PROGRAM PRG_SFLX_NoValidationCamera
VAR
	rtrigValidCameraTrigger				: F_TRIG;
	bSideFlexValidCameraTrigger			: BOOL;

	rsSideFlexTwoOutersInAggregation	: RS;
	rsSideFlexPackToOuterProcessing		: RS;

	rtrigNewOuterArrived					: R_TRIG;
	bNewOuterIsProccesing				: BOOL;
	tonValidationTimout					: TON;
	bValidationTimeout					: BOOL;
	bValidationTimeoutReset				: BOOL;
	fbTimeoutCounter						: CTU;
	nCount									: WORD;


	fbInterimCamera					: FB_SCANNER_CameraSelect;
	(*stInterimCameraOptions			: ST_SCANNER_Options := (eScannerType := E_MV_440SR_FULL, nImageBuffer := 1, nExpectedResp := 1);*)
	fbInterimCameraEvaluation		: FB_SCANNER_Evaluation;

	nInterimCameraID					: UINT;
	bInterimCameraTrigger			: BOOL;
	fbInterimCameraOut				: FB_OUTER_InterimCameraOut;

	fbCheckForDuplicateInterim	: FB_OUTER_CheckDuplicateStatus;

	rtrigInterimCameraDone			: R_TRIG;
	bInterimCameraDone				: BOOL;
	bDataReadyForValidation			: BOOL;
	bQAReject							: BOOL;

	sLastImageLableString				: T_OUTER_Barcode;

	fbPerformance							: FB_Interval;
	fbMoveOuterData						: FB_OUTER_MoveOuterStatus;
	fbCompleteDataFromConfirmation	: FB_OUTER_CompleteDataFromDB_SingleCam;
	fbMETSValidateOuterForReject			: FB_OUTER_ValidateOuterForReject;
	tofValidateOuterDoneForHMI			: TOF;
	fbMasterListUpdate					: FB_OUTER_MasterListUpdate;


	stLastOuterCompleted				: ST_OUTER_Status;
	sLastReadOuterBarcode			: T_OUTER_Barcode;
	sLastReadConfPackCode1			: T_PACK_Barcode;
	nOutersCompleted					: UDINT;
	bDoneInfo							: BOOL;


	rtrigSetOuterValidationOK			: R_TRIG;
	rtrigSetOuterValidationNOK		: R_TRIG;

	rsOuterRejectStation 				: RS;
	rsOuterRejectConfirmation 		: RS;
	tonOuterRejectReset				: TON;
	tOuterRejectActivationTime		: TIME := T#500ms;

	rtrigResetValidationStatus			: R_TRIG;

	sRejectCode						: STRING(255);
	fbArchiveInvalidOuters			: FB_OUTER_ArchiveInvalidOuters;
	aReasonForReject					: ARRAY[0..50] OF STRING(255);
	bClearList							: BOOL;

	fbOuterProduced					: FB_KPI_GenericEfficiency;
	fbOuterInspection					: FB_KPI_OutersEfficiency;

	fbOuterLevelCounter				: FB_KPI_OuterLevelCounter;

	fbQARejectCounter				: FB_CTU32;
	fbOuterValidationIndexOK			: FB_CTU32;

	ctuConsecutiveOuterRejects		: CTU;
	nActualCount						: WORD;
END_VAR
VAR // added by the converter: edge detectors and wires of the graphical bodies
    _w1, _w2 : BOOL;
END_VAR

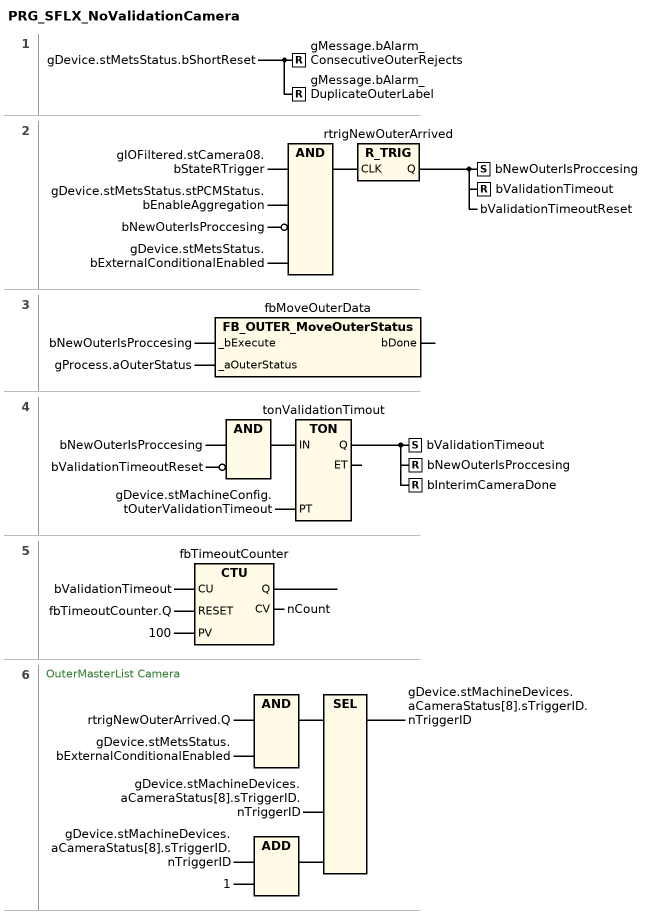
// NETWORK 1
gMessage.bAlarm_ConsecutiveOuterRejects R= gDevice.stMetsStatus.bShortReset;
gMessage.bAlarm_DuplicateOuterLabel R= gDevice.stMetsStatus.bShortReset;

// NETWORK 2
rtrigNewOuterArrived(CLK := gIOFiltered.stCamera08.bStateRTrigger AND gDevice.stMetsStatus.stPCMStatus.bEnableAggregation AND NOT bNewOuterIsProccesing AND gDevice.stMetsStatus.bExternalConditionalEnabled); // R_TRIG
bNewOuterIsProccesing S= rtrigNewOuterArrived.Q;
bValidationTimeout R= rtrigNewOuterArrived.Q;
bValidationTimeoutReset := rtrigNewOuterArrived.Q;

// NETWORK 3
fbMoveOuterData(_bExecute := bNewOuterIsProccesing, _aOuterStatus := gProcess.aOuterStatus); // FB_OUTER_MoveOuterStatus

// NETWORK 4
tonValidationTimout(IN := bNewOuterIsProccesing AND NOT bValidationTimeoutReset, PT := gDevice.stMachineConfig.tOuterValidationTimeout); // TON
bValidationTimeout S= tonValidationTimout.Q;
bNewOuterIsProccesing R= tonValidationTimout.Q;
bInterimCameraDone R= tonValidationTimout.Q;

// NETWORK 5
fbTimeoutCounter(CU := bValidationTimeout, RESET := fbTimeoutCounter.Q, PV := 100, CV => nCount); // CTU

// NETWORK 6
// OuterMasterList Camera
gDevice.stMachineDevices.aCameraStatus[8].sTriggerID.nTriggerID := SEL(rtrigNewOuterArrived.Q AND gDevice.stMetsStatus.bExternalConditionalEnabled, gDevice.stMachineDevices.aCameraStatus[8].sTriggerID.nTriggerID, gDevice.stMachineDevices.aCameraStatus[8].sTriggerID.nTriggerID + 1);

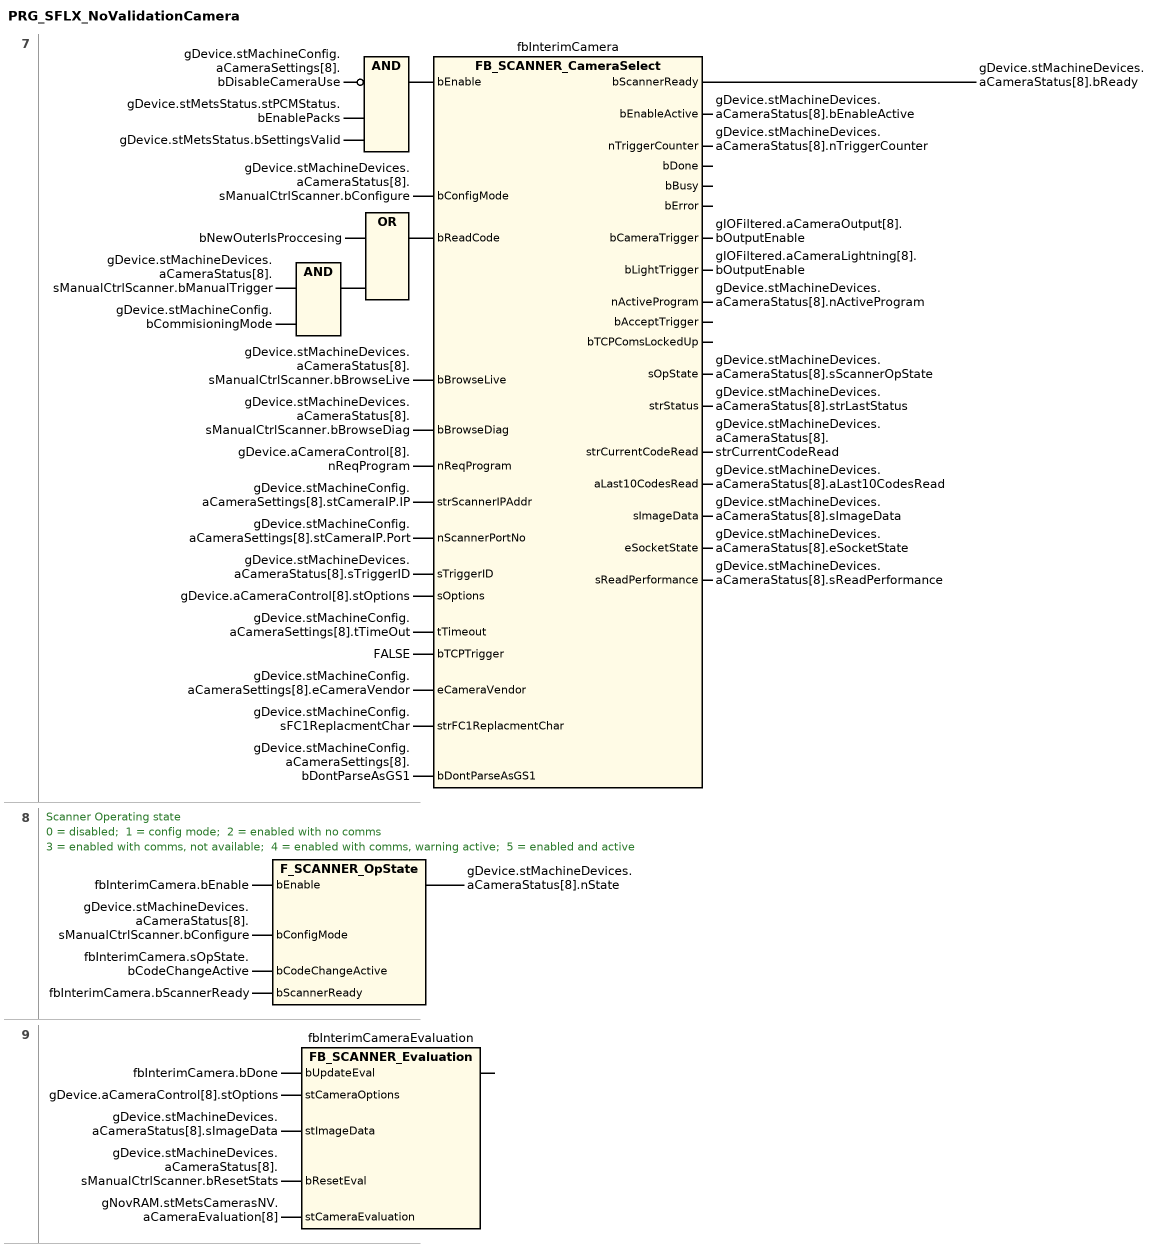
// NETWORK 7
fbInterimCamera(
    bEnable := NOT gDevice.stMachineConfig.aCameraSettings[8].bDisableCameraUse AND gDevice.stMetsStatus.stPCMStatus.bEnablePacks AND gDevice.stMetsStatus.bSettingsValid,
    bConfigMode := gDevice.stMachineDevices.aCameraStatus[8].sManualCtrlScanner.bConfigure,
    bReadCode := bNewOuterIsProccesing OR gDevice.stMachineDevices.aCameraStatus[8].sManualCtrlScanner.bManualTrigger AND gDevice.stMachineConfig.bCommisioningMode,
    bBrowseLive := gDevice.stMachineDevices.aCameraStatus[8].sManualCtrlScanner.bBrowseLive,
    bBrowseDiag := gDevice.stMachineDevices.aCameraStatus[8].sManualCtrlScanner.bBrowseDiag,
    nReqProgram := gDevice.aCameraControl[8].nReqProgram,
    strScannerIPAddr := gDevice.stMachineConfig.aCameraSettings[8].stCameraIP.IP,
    nScannerPortNo := gDevice.stMachineConfig.aCameraSettings[8].stCameraIP.Port,
    sTriggerID := gDevice.stMachineDevices.aCameraStatus[8].sTriggerID,
    sOptions := gDevice.aCameraControl[8].stOptions,
    tTimeout := gDevice.stMachineConfig.aCameraSettings[8].tTimeOut,
    bTCPTrigger := FALSE,
    eCameraVendor := gDevice.stMachineConfig.aCameraSettings[8].eCameraVendor,
    strFC1ReplacmentChar := gDevice.stMachineConfig.sFC1ReplacmentChar,
    bDontParseAsGS1 := gDevice.stMachineConfig.aCameraSettings[8].bDontParseAsGS1,
    bEnableActive => gDevice.stMachineDevices.aCameraStatus[8].bEnableActive,
    nTriggerCounter => gDevice.stMachineDevices.aCameraStatus[8].nTriggerCounter,
    bCameraTrigger => gIOFiltered.aCameraOutput[8].bOutputEnable,
    bLightTrigger => gIOFiltered.aCameraLightning[8].bOutputEnable,
    nActiveProgram => gDevice.stMachineDevices.aCameraStatus[8].nActiveProgram,
    sOpState => gDevice.stMachineDevices.aCameraStatus[8].sScannerOpState,
    strStatus => gDevice.stMachineDevices.aCameraStatus[8].strLastStatus,
    strCurrentCodeRead => gDevice.stMachineDevices.aCameraStatus[8].strCurrentCodeRead,
    aLast10CodesRead => gDevice.stMachineDevices.aCameraStatus[8].aLast10CodesRead,
    sImageData => gDevice.stMachineDevices.aCameraStatus[8].sImageData,
    eSocketState => gDevice.stMachineDevices.aCameraStatus[8].eSocketState,
    sReadPerformance => gDevice.stMachineDevices.aCameraStatus[8].sReadPerformance); // FB_SCANNER_CameraSelect
gDevice.stMachineDevices.aCameraStatus[8].bReady := fbInterimCamera.bScannerReady;

// NETWORK 8
// 					Scanner Operating state
// 0 = disabled;  1 = config mode;  2 = enabled with no comms
// 3 = enabled with comms, not available;  4 = enabled with comms, warning active;  5 = enabled and active
//
gDevice.stMachineDevices.aCameraStatus[8].nState := F_SCANNER_OpState(bEnable := fbInterimCamera.bEnable, bConfigMode := gDevice.stMachineDevices.aCameraStatus[8].sManualCtrlScanner.bConfigure, bCodeChangeActive := fbInterimCamera.sOpState.bCodeChangeActive, bScannerReady := fbInterimCamera.bScannerReady);

// NETWORK 9
fbInterimCameraEvaluation(
    bUpdateEval := fbInterimCamera.bDone,
    stCameraOptions := gDevice.aCameraControl[8].stOptions,
    stImageData := gDevice.stMachineDevices.aCameraStatus[8].sImageData,
    bResetEval := gDevice.stMachineDevices.aCameraStatus[8].sManualCtrlScanner.bResetStats,
    stCameraEvaluation := gNovRAM.stMetsCamerasNV.aCameraEvaluation[8]); // FB_SCANNER_Evaluation

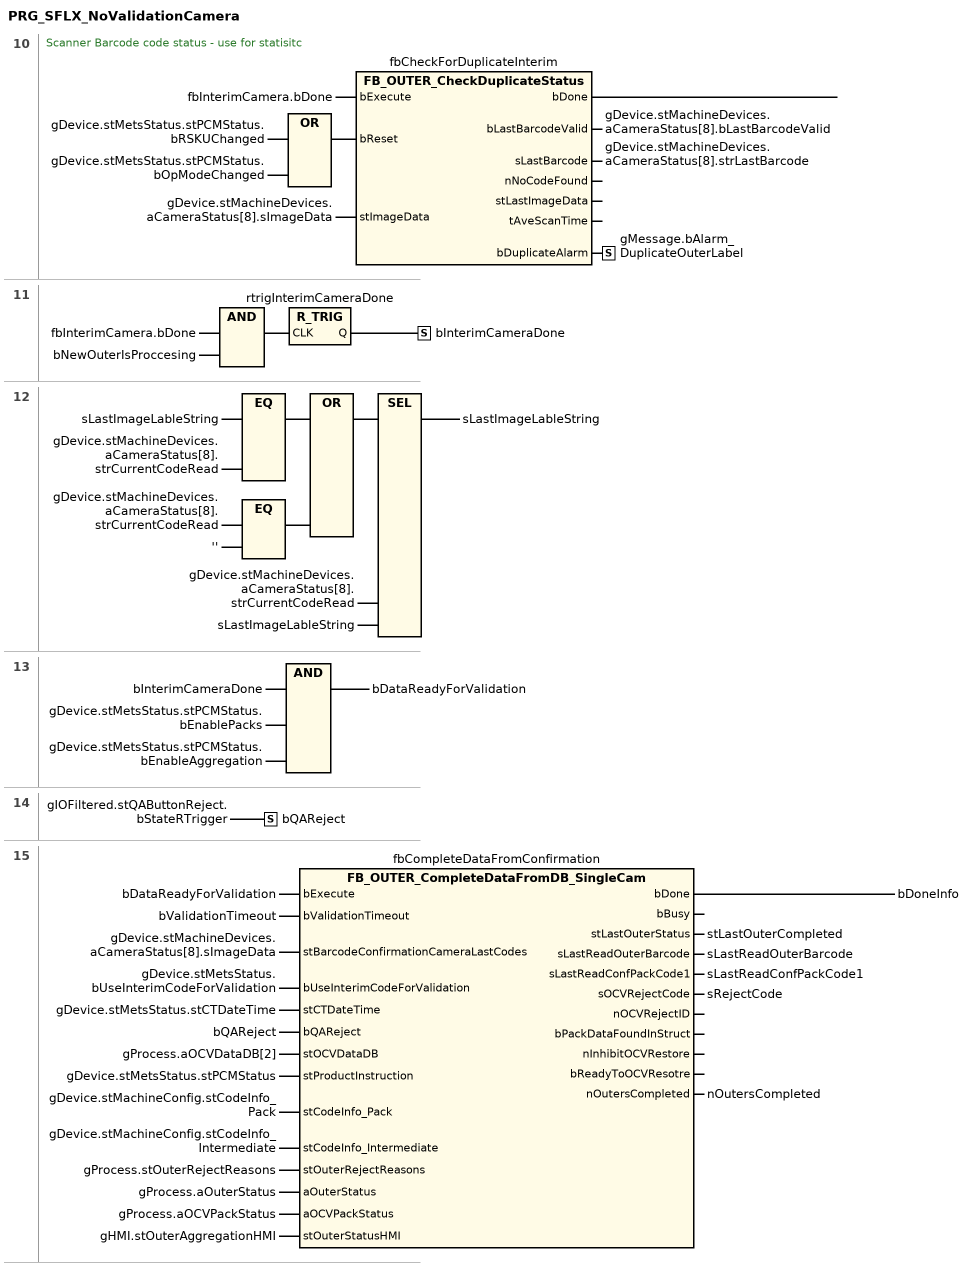
// NETWORK 10
// Scanner Barcode code status - use for statisitc
fbCheckForDuplicateInterim(
    bExecute := fbInterimCamera.bDone,
    bReset := gDevice.stMetsStatus.stPCMStatus.bRSKUChanged OR gDevice.stMetsStatus.stPCMStatus.bOpModeChanged,
    stImageData := gDevice.stMachineDevices.aCameraStatus[8].sImageData,
    bLastBarcodeValid => gDevice.stMachineDevices.aCameraStatus[8].bLastBarcodeValid,
    sLastBarcode => gDevice.stMachineDevices.aCameraStatus[8].strLastBarcode); // FB_OUTER_CheckDuplicateStatus
gMessage.bAlarm_DuplicateOuterLabel S= fbCheckForDuplicateInterim.bDuplicateAlarm;

// NETWORK 11
rtrigInterimCameraDone(CLK := fbInterimCamera.bDone AND bNewOuterIsProccesing); // R_TRIG
bInterimCameraDone S= rtrigInterimCameraDone.Q;

// NETWORK 12
sLastImageLableString := SEL(sLastImageLableString = gDevice.stMachineDevices.aCameraStatus[8].strCurrentCodeRead OR gDevice.stMachineDevices.aCameraStatus[8].strCurrentCodeRead = '', gDevice.stMachineDevices.aCameraStatus[8].strCurrentCodeRead, sLastImageLableString);

// NETWORK 13
bDataReadyForValidation := bInterimCameraDone AND gDevice.stMetsStatus.stPCMStatus.bEnablePacks AND gDevice.stMetsStatus.stPCMStatus.bEnableAggregation;

// NETWORK 14
bQAReject S= gIOFiltered.stQAButtonReject.bStateRTrigger;

// NETWORK 15
fbCompleteDataFromConfirmation(
    bExecute := bDataReadyForValidation,
    bValidationTimeout := bValidationTimeout,
    stBarcodeConfirmationCameraLastCodes := gDevice.stMachineDevices.aCameraStatus[8].sImageData,
    bUseInterimCodeForValidation := gDevice.stMetsStatus.bUseInterimCodeForValidation,
    stCTDateTime := gDevice.stMetsStatus.stCTDateTime,
    bQAReject := bQAReject,
    stOCVDataDB := gProcess.aOCVDataDB[2],
    stProductInstruction := gDevice.stMetsStatus.stPCMStatus,
    stCodeInfo_Pack := gDevice.stMachineConfig.stCodeInfo_Pack,
    stCodeInfo_Intermediate := gDevice.stMachineConfig.stCodeInfo_Intermediate,
    stOuterRejectReasons := gProcess.stOuterRejectReasons,
    aOuterStatus := gProcess.aOuterStatus,
    aOCVPackStatus := gProcess.aOCVPackStatus,
    stOuterStatusHMI := gHMI.stOuterAggregationHMI,
    stLastOuterStatus => stLastOuterCompleted,
    sLastReadOuterBarcode => sLastReadOuterBarcode,
    sLastReadConfPackCode1 => sLastReadConfPackCode1,
    sOCVRejectCode => sRejectCode,
    nOutersCompleted => nOutersCompleted); // FB_OUTER_CompleteDataFromDB_SingleCam
bDoneInfo := fbCompleteDataFromConfirmation.bDone;

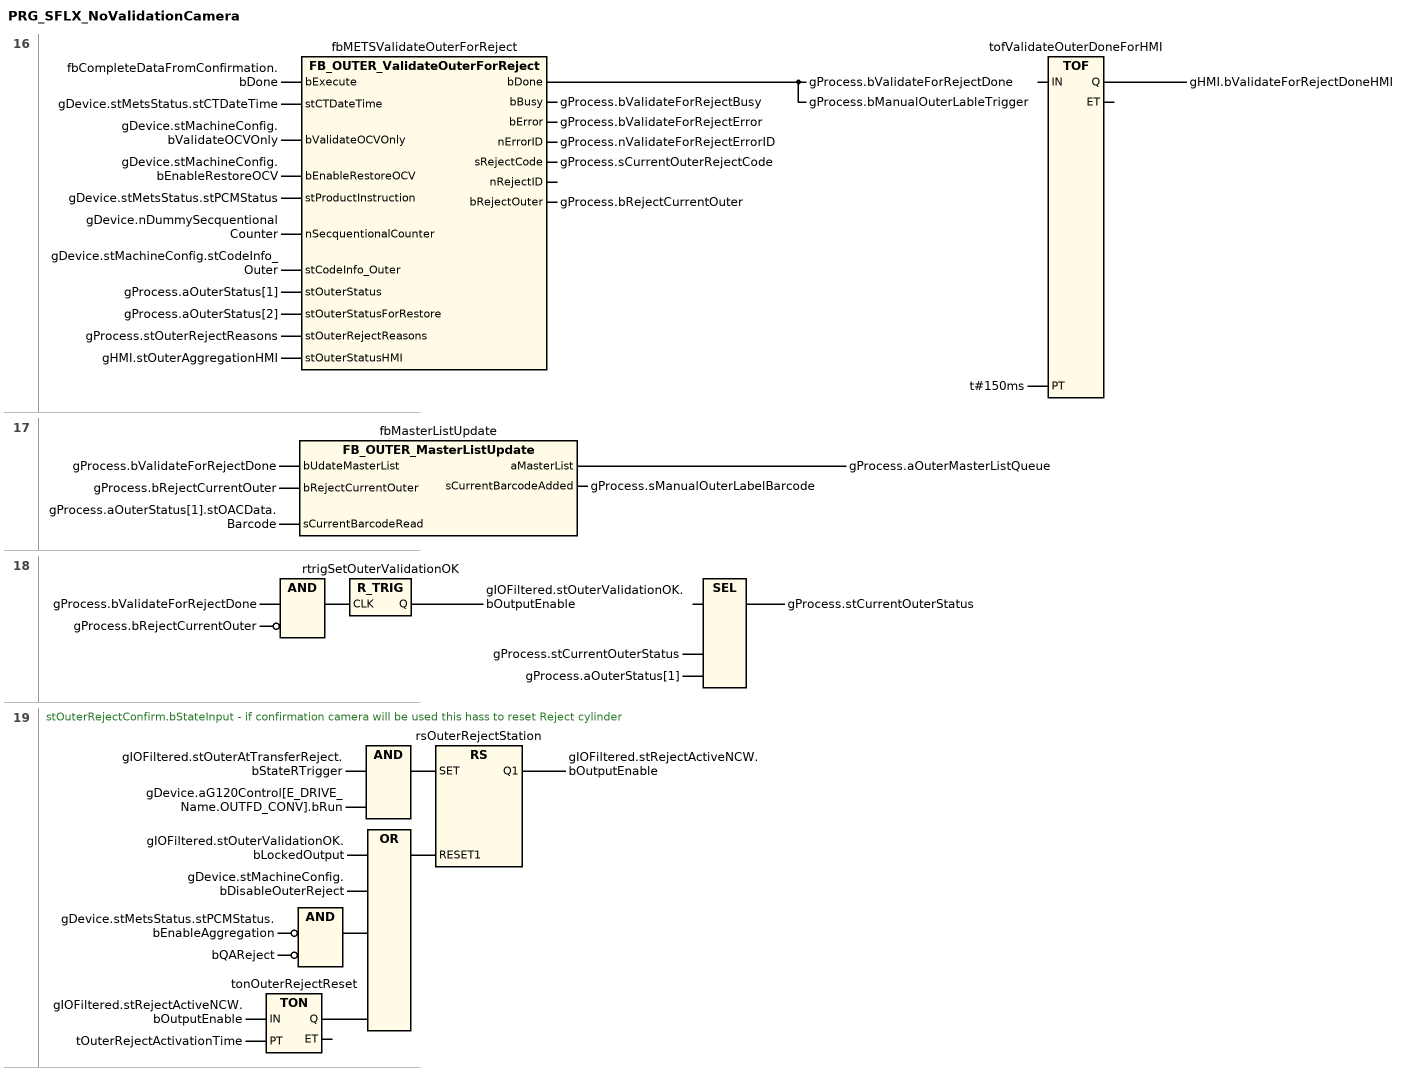
// NETWORK 16
fbMETSValidateOuterForReject(
    bExecute := fbCompleteDataFromConfirmation.bDone,
    stCTDateTime := gDevice.stMetsStatus.stCTDateTime,
    bValidateOCVOnly := gDevice.stMachineConfig.bValidateOCVOnly,
    bEnableRestoreOCV := gDevice.stMachineConfig.bEnableRestoreOCV,
    stProductInstruction := gDevice.stMetsStatus.stPCMStatus,
    nSecquentionalCounter := gDevice.nDummySecquentionalCounter,
    stCodeInfo_Outer := gDevice.stMachineConfig.stCodeInfo_Outer,
    stOuterStatus := gProcess.aOuterStatus[1],
    stOuterStatusForRestore := gProcess.aOuterStatus[2],
    stOuterRejectReasons := gProcess.stOuterRejectReasons,
    stOuterStatusHMI := gHMI.stOuterAggregationHMI,
    bBusy => gProcess.bValidateForRejectBusy,
    bError => gProcess.bValidateForRejectError,
    nErrorID => gProcess.nValidateForRejectErrorID,
    sRejectCode => gProcess.sCurrentOuterRejectCode,
    bRejectOuter => gProcess.bRejectCurrentOuter); // FB_OUTER_ValidateOuterForReject
gProcess.bValidateForRejectDone := fbMETSValidateOuterForReject.bDone;
gProcess.bManualOuterLableTrigger := fbMETSValidateOuterForReject.bDone;
tofValidateOuterDoneForHMI(IN := fbMETSValidateOuterForReject.bDone, PT := t#150ms); // TOF
gHMI.bValidateForRejectDoneHMI := tofValidateOuterDoneForHMI.Q;

// NETWORK 17
fbMasterListUpdate(
    bUdateMasterList := gProcess.bValidateForRejectDone,
    bRejectCurrentOuter := gProcess.bRejectCurrentOuter,
    sCurrentBarcodeRead := gProcess.aOuterStatus[1].stOACData.Barcode,
    sCurrentBarcodeAdded => gProcess.sManualOuterLabelBarcode); // FB_OUTER_MasterListUpdate
gProcess.aOuterMasterListQueue := fbMasterListUpdate.aMasterList;

// NETWORK 18
rtrigSetOuterValidationOK(CLK := gProcess.bValidateForRejectDone AND NOT gProcess.bRejectCurrentOuter); // R_TRIG
gIOFiltered.stOuterValidationOK.bOutputEnable := rtrigSetOuterValidationOK.Q;
gProcess.stCurrentOuterStatus := SEL(rtrigSetOuterValidationOK.Q, gProcess.stCurrentOuterStatus, gProcess.aOuterStatus[1]);

// NETWORK 19
// stOuterRejectConfirm.bStateInput - if confirmation camera will be used this hass to reset Reject cylinder
tonOuterRejectReset(IN := gIOFiltered.stRejectActiveNCW.bOutputEnable, PT := tOuterRejectActivationTime); // TON
rsOuterRejectStation(SET := gIOFiltered.stOuterAtTransferReject.bStateRTrigger AND gDevice.aG120Control[E_DRIVE_Name.OUTFD_CONV].bRun, RESET1 := gIOFiltered.stOuterValidationOK.bLockedOutput OR gDevice.stMachineConfig.bDisableOuterReject OR NOT gDevice.stMetsStatus.stPCMStatus.bEnableAggregation AND NOT bQAReject OR tonOuterRejectReset.Q); // RS
gIOFiltered.stRejectActiveNCW.bOutputEnable := rsOuterRejectStation.Q1;

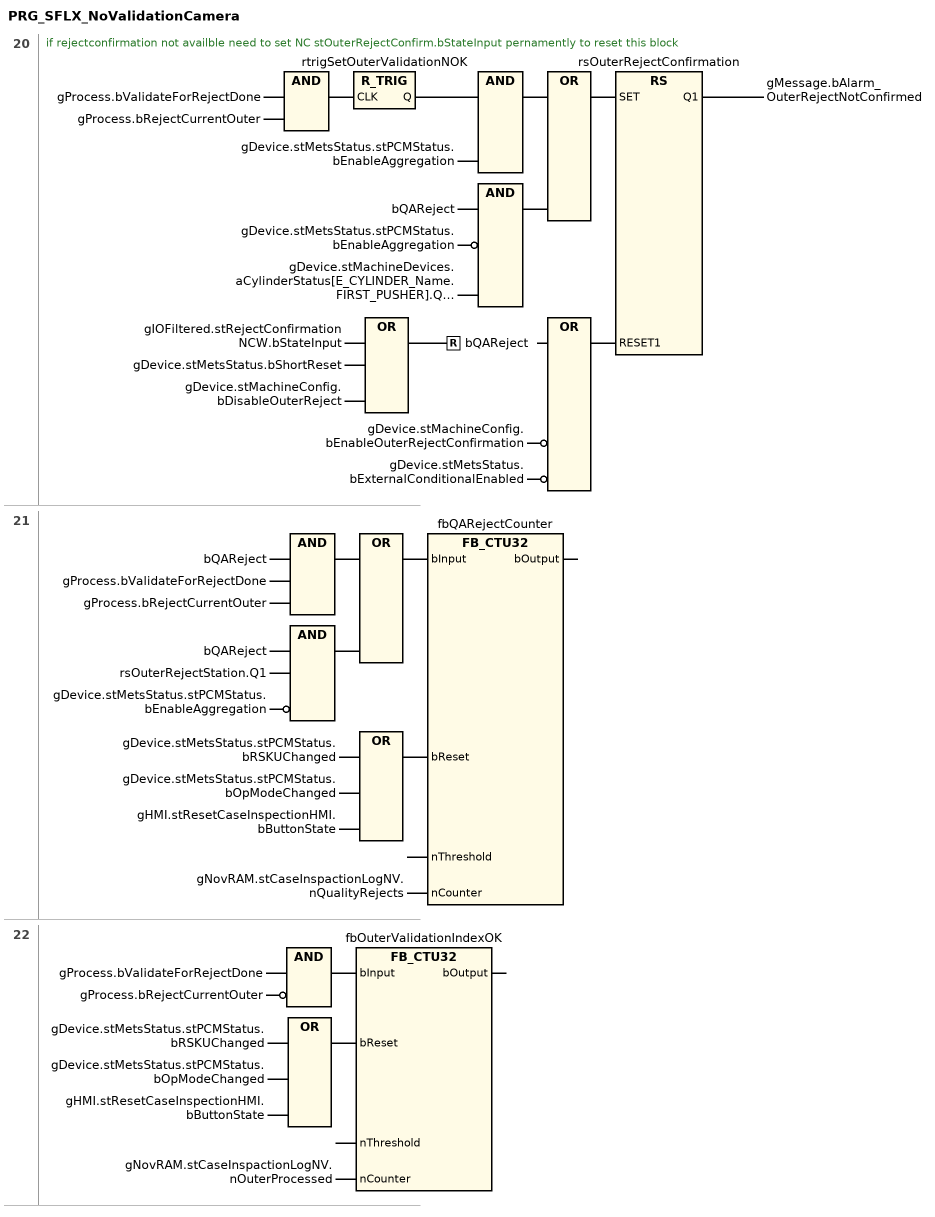
// NETWORK 20
// if rejectconfirmation not availble need to set NC stOuterRejectConfirm.bStateInput pernamently to reset this block
rtrigSetOuterValidationNOK(CLK := gProcess.bValidateForRejectDone AND gProcess.bRejectCurrentOuter); // R_TRIG
_w2 := rtrigSetOuterValidationNOK.Q AND gDevice.stMetsStatus.stPCMStatus.bEnableAggregation OR bQAReject AND NOT gDevice.stMetsStatus.stPCMStatus.bEnableAggregation AND gDevice.stMachineDevices.aCylinderStatus[E_CYLINDER_Name.FIRST_PUSHER].Q.bCylinderInExtendedPosition;
_w1 := gIOFiltered.stRejectConfirmationNCW.bStateInput OR gDevice.stMetsStatus.bShortReset OR gDevice.stMachineConfig.bDisableOuterReject;
bQAReject R= _w1;
rsOuterRejectConfirmation(SET := _w2, RESET1 := _w1 OR NOT gDevice.stMachineConfig.bEnableOuterRejectConfirmation OR NOT gDevice.stMetsStatus.bExternalConditionalEnabled); // RS
gMessage.bAlarm_OuterRejectNotConfirmed := rsOuterRejectConfirmation.Q1;

// NETWORK 21
fbQARejectCounter(
    bInput := bQAReject AND gProcess.bValidateForRejectDone AND gProcess.bRejectCurrentOuter OR bQAReject AND rsOuterRejectStation.Q1 AND NOT gDevice.stMetsStatus.stPCMStatus.bEnableAggregation,
    bReset := gDevice.stMetsStatus.stPCMStatus.bRSKUChanged OR gDevice.stMetsStatus.stPCMStatus.bOpModeChanged OR gHMI.stResetCaseInspectionHMI.bButtonState,
    nCounter := gNovRAM.stCaseInspactionLogNV.nQualityRejects); // FB_CTU32

// NETWORK 22
fbOuterValidationIndexOK(
    bInput := gProcess.bValidateForRejectDone AND NOT gProcess.bRejectCurrentOuter,
    bReset := gDevice.stMetsStatus.stPCMStatus.bRSKUChanged OR gDevice.stMetsStatus.stPCMStatus.bOpModeChanged OR gHMI.stResetCaseInspectionHMI.bButtonState,
    nCounter := gNovRAM.stCaseInspactionLogNV.nOuterProcessed); // FB_CTU32

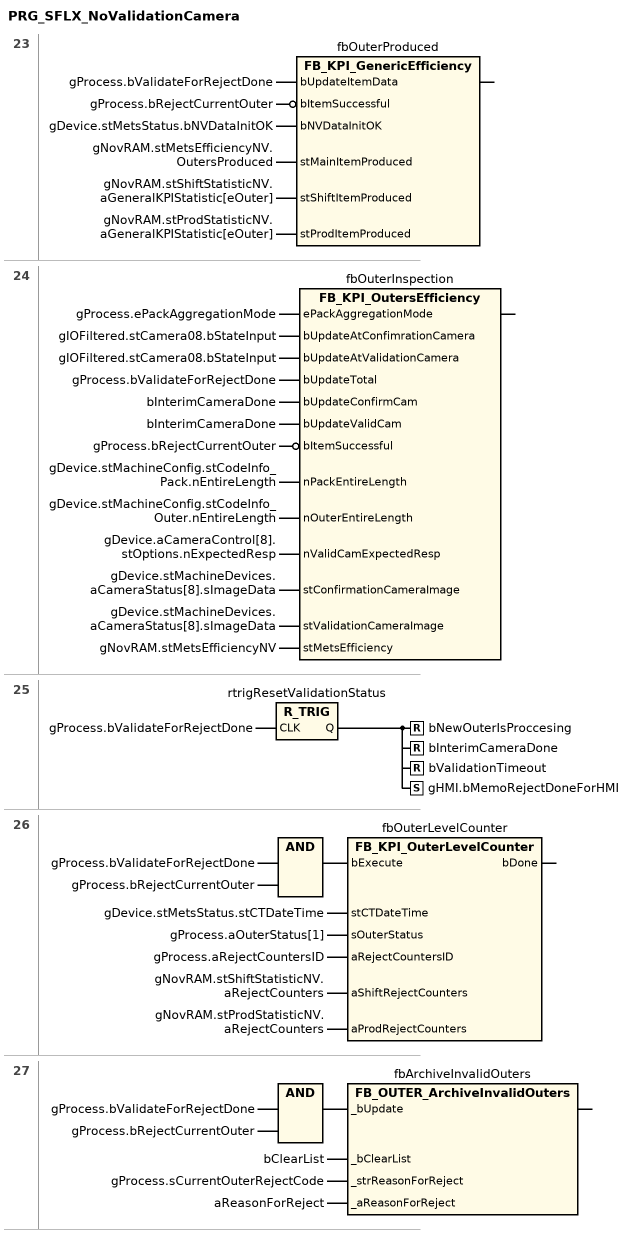
// NETWORK 23
fbOuterProduced(
    bUpdateItemData := gProcess.bValidateForRejectDone,
    bItemSuccessful := NOT gProcess.bRejectCurrentOuter,
    bNVDataInitOK := gDevice.stMetsStatus.bNVDataInitOK,
    stMainItemProduced := gNovRAM.stMetsEfficiencyNV.OutersProduced,
    stShiftItemProduced := gNovRAM.stShiftStatisticNV.aGeneralKPIStatistic[eOuter],
    stProdItemProduced := gNovRAM.stProdStatisticNV.aGeneralKPIStatistic[eOuter]); // FB_KPI_GenericEfficiency

// NETWORK 24
fbOuterInspection(
    ePackAggregationMode := gProcess.ePackAggregationMode,
    bUpdateAtConfimrationCamera := gIOFiltered.stCamera08.bStateInput,
    bUpdateAtValidationCamera := gIOFiltered.stCamera08.bStateInput,
    bUpdateTotal := gProcess.bValidateForRejectDone,
    bUpdateConfirmCam := bInterimCameraDone,
    bUpdateValidCam := bInterimCameraDone,
    bItemSuccessful := NOT gProcess.bRejectCurrentOuter,
    nPackEntireLength := gDevice.stMachineConfig.stCodeInfo_Pack.nEntireLength,
    nOuterEntireLength := gDevice.stMachineConfig.stCodeInfo_Outer.nEntireLength,
    nValidCamExpectedResp := gDevice.aCameraControl[8].stOptions.nExpectedResp,
    stConfirmationCameraImage := gDevice.stMachineDevices.aCameraStatus[8].sImageData,
    stValidationCameraImage := gDevice.stMachineDevices.aCameraStatus[8].sImageData,
    stMetsEfficiency := gNovRAM.stMetsEfficiencyNV); // FB_KPI_OutersEfficiency

// NETWORK 25
rtrigResetValidationStatus(CLK := gProcess.bValidateForRejectDone); // R_TRIG
bNewOuterIsProccesing R= rtrigResetValidationStatus.Q;
bInterimCameraDone R= rtrigResetValidationStatus.Q;
bValidationTimeout R= rtrigResetValidationStatus.Q;
gHMI.bMemoRejectDoneForHMI S= rtrigResetValidationStatus.Q;

// NETWORK 26
fbOuterLevelCounter(
    bExecute := gProcess.bValidateForRejectDone AND gProcess.bRejectCurrentOuter,
    stCTDateTime := gDevice.stMetsStatus.stCTDateTime,
    sOuterStatus := gProcess.aOuterStatus[1],
    aRejectCountersID := gProcess.aRejectCountersID,
    aShiftRejectCounters := gNovRAM.stShiftStatisticNV.aRejectCounters,
    aProdRejectCounters := gNovRAM.stProdStatisticNV.aRejectCounters); // FB_KPI_OuterLevelCounter

// NETWORK 27
fbArchiveInvalidOuters(
    _bUpdate := gProcess.bValidateForRejectDone AND gProcess.bRejectCurrentOuter,
    _bClearList := bClearList,
    _strReasonForReject := gProcess.sCurrentOuterRejectCode,
    _aReasonForReject := aReasonForReject); // FB_OUTER_ArchiveInvalidOuters

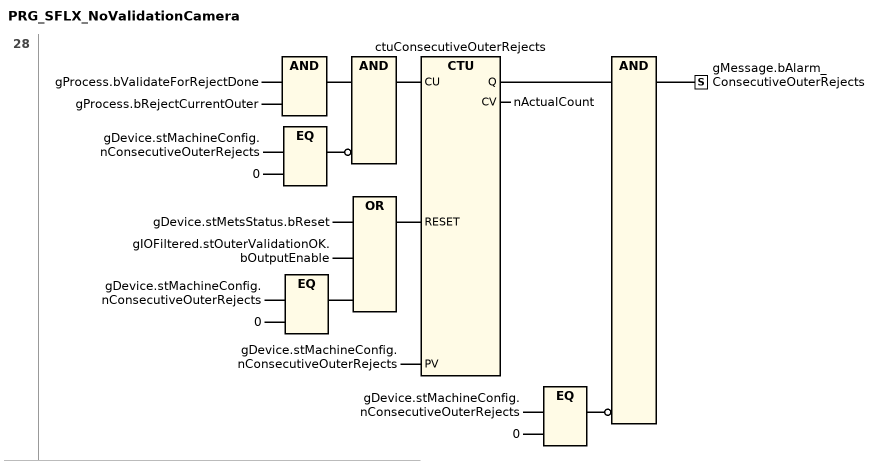
// NETWORK 28
ctuConsecutiveOuterRejects(
    CU := (gProcess.bValidateForRejectDone AND gProcess.bRejectCurrentOuter) AND NOT (gDevice.stMachineConfig.nConsecutiveOuterRejects = 0),
    RESET := gDevice.stMetsStatus.bReset OR gIOFiltered.stOuterValidationOK.bOutputEnable OR gDevice.stMachineConfig.nConsecutiveOuterRejects = 0,
    PV := gDevice.stMachineConfig.nConsecutiveOuterRejects,
    CV => nActualCount); // CTU
gMessage.bAlarm_ConsecutiveOuterRejects S= ctuConsecutiveOuterRejects.Q AND NOT (gDevice.stMachineConfig.nConsecutiveOuterRejects = 0);

END_PROGRAM

(* stored: Version 1.1.0.1
   POU PRG_SFLX_NoValidationCamera: Id {177ef6c9-4a7c-4528-ac8c-d9896912667b}, SpecialFunc None *)
